FUNCTION_BLOCK POU3
VAR_INPUT
END_VAR
VAR_OUTPUT
END_VAR
VAR
END_VAR

END_FUNCTION_BLOCK

(* stored: Version 1.1.0.1, ProductVersion 3.1.4020.12
   POU POU3: Id {43eb077f-1080-4cfa-95d4-aac7502529e3}, SpecialFunc None *)
